FUNCTION_BLOCK FB_ExampleCow
VAR_INPUT
END_VAR
VAR_OUTPUT
END_VAR
VAR
END_VAR

END_FUNCTION_BLOCK

(* stored: Version 1.1.0.1, ProductVersion 3.1.4022.18
   POU FB_ExampleCow: Id {d8a4f85f-5611-4e0a-b457-d3ba5721fd09}, SpecialFunc None *)
